(* PLC project Beremiz Python Support Tests, Beremiz 0.0 *)
(* stored: creationDateTime 2008-12-14T16:21:19, contentDescription This example shows many features in Beremiz: 1. How to implement python extensions. 2. How to implement basic C extension. 3. How to use C code in IEC POUs. 4. How to call C functions from python code. 5. How to avoid race conditions between IEC, C and python code. 6. How to convert betweet different IEC types., modificationDateTime 2018-09-26T13:15:28 *)

TYPE CPLX_TYPE : STRUCT
  FIRSTBYTE : SINT;
  SECONDBYTE : SINT;
END_STRUCT;
END_TYPE

TYPE StateMachine : (STANDBY, START, STOP);
END_TYPE

TYPE datatype0 : BOOL;
END_TYPE

FUNCTION_BLOCK C_Pragma
  VAR_OUTPUT
    OUT : SINT;
  END_VAR
  VAR_INPUT
    IN : SINT;
  END_VAR
  VAR
    COORDS : ARRAY[0..5] OF SINT := [54, 55, 56, 57, 58, 59];
    SMURF : CPLX_TYPE;
  END_VAR
  VAR_EXTERNAL
    Global_RS : RS;
  END_VAR

            (* hereafter is a C pragma accessing FB interface in a clean way *)
{{
  char toPLC;
  char fromPLC = GetFbVar(IN);
  extern int PLC_C_Call(char, char *);
  if(PLC_C_Call(fromPLC, &toPLC)){
    SetFbVar(OUT, toPLC);
  }
  if(0){
    /* that code demonstrate C access to complex types */
    char somebyte = GetFbVar(COORDS, .table[3]);
    SetFbVar(SMURF, somebyte, .FIRSTBYTE);
    SetFbVar(COORDS, somebyte, .table[4]);
  }
}}
(* If you do not use GetFbVar and SetFbVar macros, expect unexpected behaviour*)
Global_RS();

          
END_FUNCTION_BLOCK

FUNCTION function0 : datatype0
  VAR_INPUT
    LocalVar0 : datatype0;
  END_VAR

            function0 := LocalVar0;

          
END_FUNCTION

PROGRAM main_pytest
  VAR
    mux1_sel : INT := 3;
    mux2_sel : INT := 3;
    pytest_var1 : STRING;
    fefvsd : datatype0;
    pytest_var2 : BOOL;
    py1 : python_eval;
    Block1 : python_eval;
    Block2 : python_eval;
    Block3 : python_eval;
    pytest_var3 : BOOL;
    FromC : SINT;
    C_Pragma0 : C_Pragma;
  END_VAR
  VAR_EXTERNAL
    TestInput : SINT;
    TestOutput : SINT;
  END_VAR
  VAR
    FromInput : SINT;
    Test_BCD : WORD := 151;
    Test_BCD_WRONG : WORD := 154;
    Test_BCD_CONVERTED : BOOL;
    Test_BCD_RESULT : UINT;
    Test_BCD_WRONG_RESULT : UINT;
    Test_DT : DT := DT#2013-02-23-22:35:46;
    Test_TOD : TOD;
    Test_TOD_STRING : STRING;
    Test_Date : DATE;
    Test_String : STRING := 'test';
    Test_Bool : BOOL;
  END_VAR
  VAR_EXTERNAL
    Global_RS : RS;
    TUTU : INT;
    TOTO : INT;
    Test_Python_Var : INT;
    Second_Python_Var : INT;
  END_VAR
  VAR  (* added by the conversion: wires and edge detectors of the diagram *)
    _NOT7_OUT : BOOL;
  END_VAR

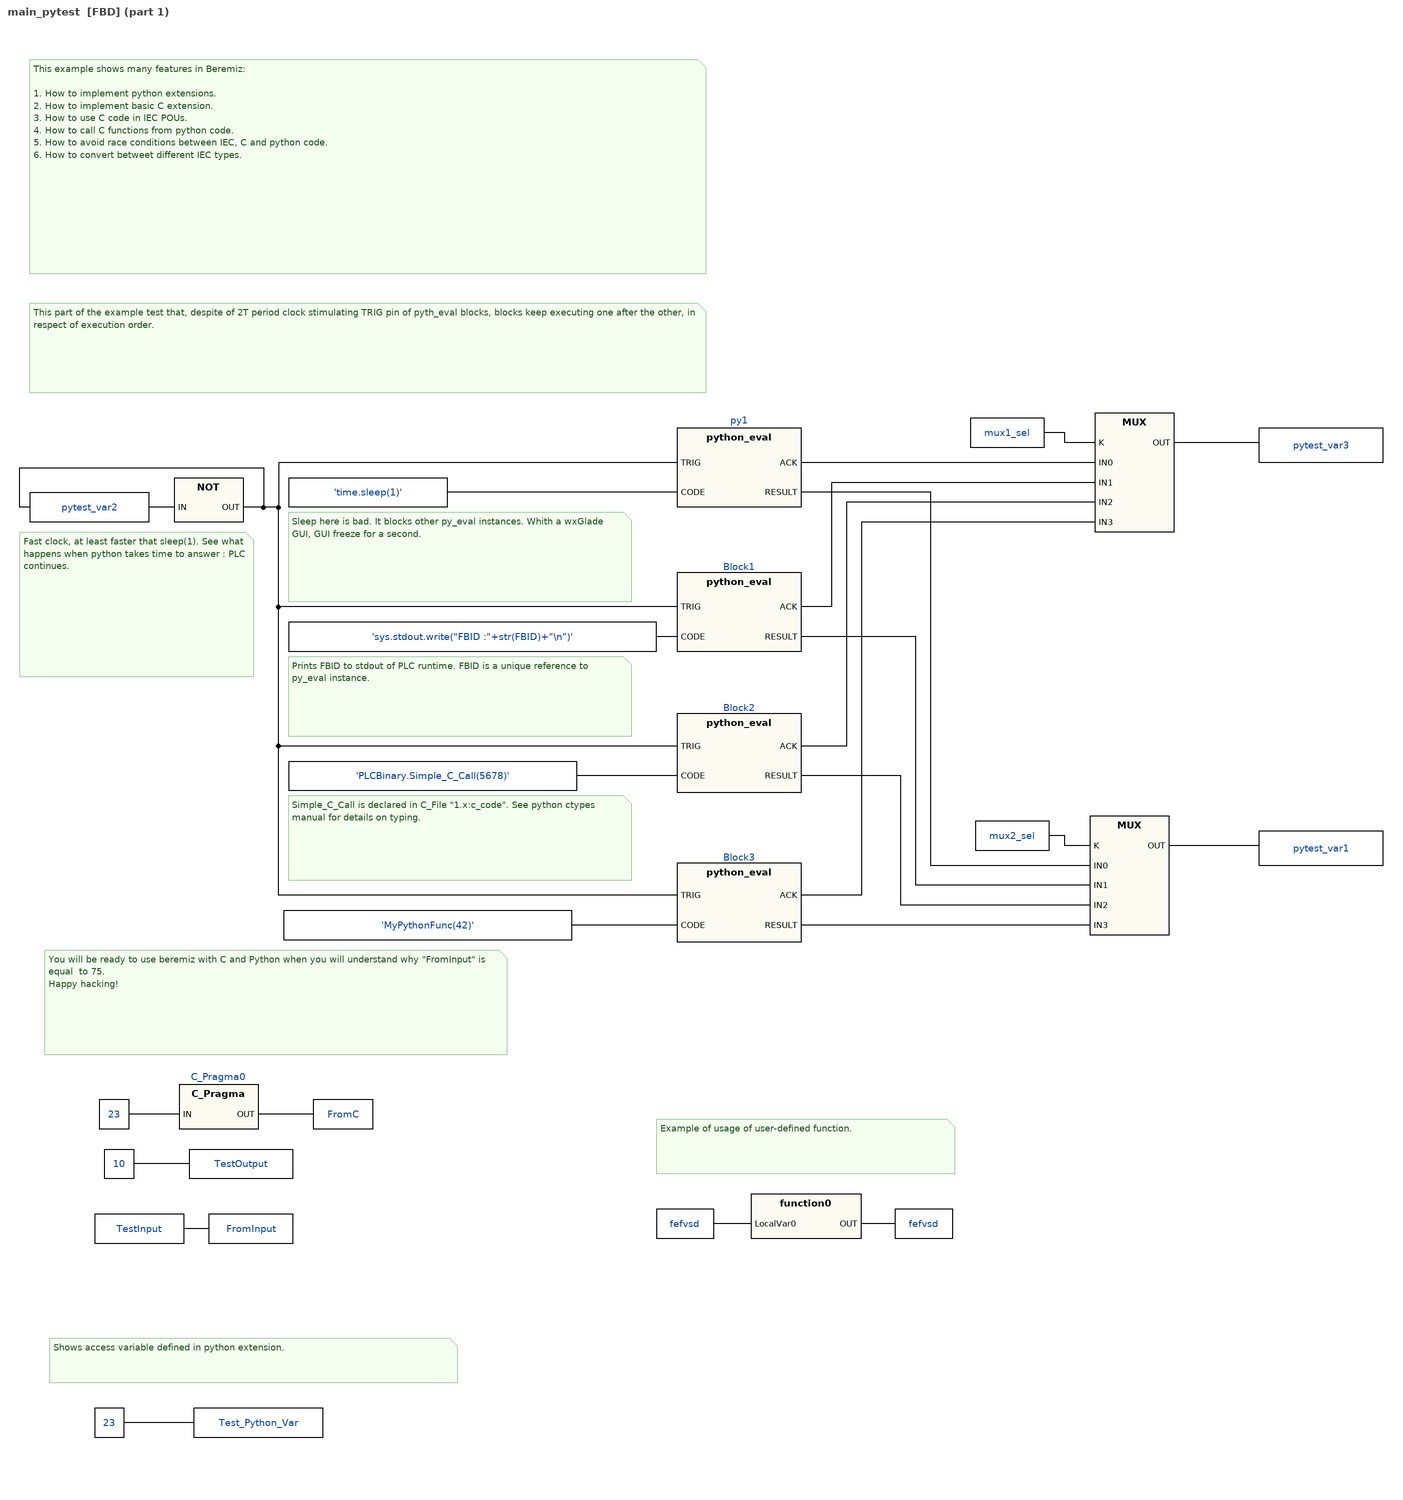
(* FBD diagram, written out as Structured Text *)
(* This example shows many features in Beremiz:

   1. How to implement python extensions.
   2. How to implement basic C extension.
   3. How to use C code in IEC POUs.
   4. How to call C functions from python code.
   5. How to avoid race conditions between IEC, C and python code.
   6. How to convert betweet different IEC types. *)
(* This part of the example test that, despite of 2T period clock stimulating TRIG pin of pyth_eval blocks, blocks keep executing one after the other, in respect of execution order. *)
_NOT7_OUT := NOT pytest_var2;
py1(TRIG := _NOT7_OUT, CODE := 'time.sleep(1)');
Block1(TRIG := _NOT7_OUT, CODE := 'sys.stdout.write("FBID :"+str(FBID)+"\n")');
Block2(TRIG := _NOT7_OUT, CODE := 'PLCBinary.Simple_C_Call(5678)');
Block3(TRIG := _NOT7_OUT, CODE := 'MyPythonFunc(42)');
pytest_var3 := MUX(mux1_sel, py1.ACK, Block1.ACK, Block2.ACK, Block3.ACK);
pytest_var2 := _NOT7_OUT;
(* Sleep here is bad. It blocks other py_eval instances. Whith a wxGlade GUI, GUI freeze for a second. *)
(* Fast clock, at least faster that sleep(1). See what happens when python takes time to answer : PLC continues. *)
(* Prints FBID to stdout of PLC runtime. FBID is a unique reference to py_eval instance. *)
(* Simple_C_Call is declared in C_File "1.x:c_code". See python ctypes manual for details on typing. *)
pytest_var1 := MUX(mux2_sel, py1.RESULT, Block1.RESULT, Block2.RESULT, Block3.RESULT);
(* You will be ready to use beremiz with C and Python when you will understand why "FromInput" is equal  to 75.
Happy hacking! *)
C_Pragma0(IN := 23);
FromC := C_Pragma0.OUT;
(* Example of usage of user-defined function. *)
TestOutput := 10;
FromInput := TestInput;
fefvsd := function0(fefvsd);
(* Shows access variable defined in python extension. *)
Test_Python_Var := 23;
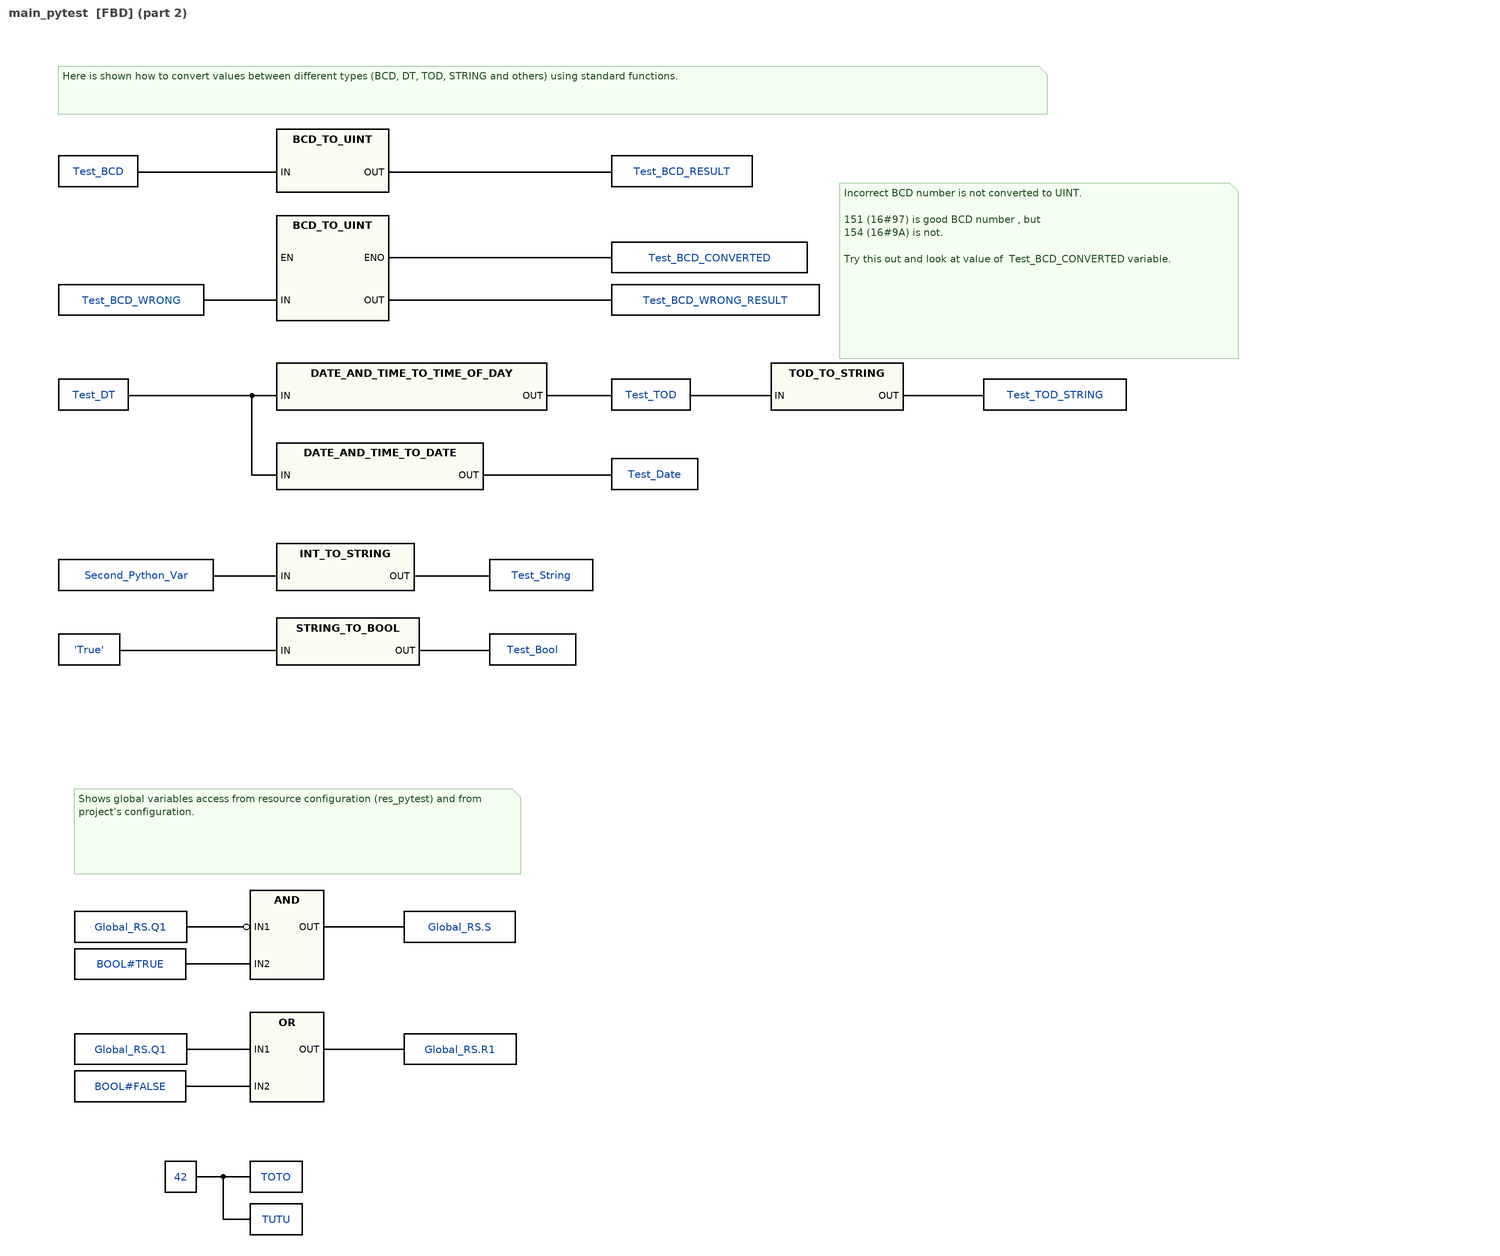
(* Here is shown how to convert values between different types (BCD, DT, TOD, STRING and others) using standard functions. *)
Test_BCD_RESULT := BCD_TO_UINT(Test_BCD);
(* Incorrect BCD number is not converted to UINT.

151 (16#97) is good BCD number , but 
154 (16#9A) is not.  

Try this out and look at value of  Test_BCD_CONVERTED variable. *)
Test_BCD_CONVERTED := TRUE;
Test_BCD_WRONG_RESULT := BCD_TO_UINT(Test_BCD_WRONG);
Test_TOD := DATE_AND_TIME_TO_TIME_OF_DAY(Test_DT);
Test_TOD_STRING := TOD_TO_STRING(Test_TOD);
Test_Date := DATE_AND_TIME_TO_DATE(Test_DT);
Test_String := INT_TO_STRING(Second_Python_Var);
Test_Bool := STRING_TO_BOOL('True');
(* Shows global variables access from resource configuration (res_pytest) and from project's configuration. *)
Global_RS.S := NOT Global_RS.Q1 AND BOOL#TRUE;
Global_RS.R1 := Global_RS.Q1 OR BOOL#FALSE;
TOTO := 42;
TUTU := 42;
END_PROGRAM

FUNCTION norm : REAL
  VAR_INPUT
    IN1 : REAL;
    IN2 : REAL;
  END_VAR

            NORM := SQRT(IN1 * IN1 + IN2 * IN2);
          
END_FUNCTION

CONFIGURATION config
  VAR_GLOBAL
    Global_RS : RS;
    TUTU : INT;
  END_VAR
  RESOURCE res_pytest ON PLC
    VAR_GLOBAL
      TOTO : INT;
    END_VAR
    TASK pytest_task(INTERVAL := T#1ms, PRIORITY := 0);
    PROGRAM pytest_instance : main_pytest;
  END_RESOURCE
END_CONFIGURATION
